(* CoDeSys 2.3 export: MNG_APPLICATION_INPUTS_32BIT.EXP *)

(* Data type *)
(*                                                                            *)

TYPE MNG_APPLICATION_INPUTS_32BIT :
STRUCT
    NumSignals                    : INT     := 0         ;
END_STRUCT
END_TYPE
